// TIA Portal V19 export
ORGANIZATION_BLOCK "RESTART"   // OB100, STL, Startup
TITLE = Start-Up
{ S7_Optimized_Access := 'TRUE' }
VERSION : 0.0
// Comment
// stored: AutoNumber false
   VAR_INPUT
      LostRetentive : Bool;   // True if retentive data are lost
      LostRTC : Bool;   // True if date and time are lost
   END_VAR
BEGIN

NETWORK
TITLE = 
      L     0;
      T     "OP25 TANK".TaTimerStep;
      T     "OP25 TANK".TaTimerActual;
      T     "OP25 TANK".TaMainUpdating;
      T     "OP25 TANK".TaStepUpdating;

NETWORK
TITLE = 
      SET;
      R     "LEDAssignment".K1_FLASH;  //"FLASH_K1_SPARE"
      R     "LEDAssignment".K1_LIGHT;  //"LIGHT_K1_SPARE"
      R     "LEDAssignment".K2_FLASH;  //"FLASH_K2_SPARE"
      R     "LEDAssignment".K2_LIGHT;  //"LIGHT_K2_SPARE"
      R     "LEDAssignment".K3_FLASH;  //"FLASH_K3_PRESTE."
      R     "LEDAssignment".K3_LIGHT;  //"LIGHT_K3_PRESTE."
      R     "LEDAssignment".K4_FLASH;  //"FLASH_K4_CIP_LYE"
      R     "LEDAssignment".K4_LIGHT;  //"LIGHT_K4_CIP_LYE"
      R     "LEDAssignment".K5_FLASH;  //"FLASH_K5_CIP_LYE_ACID"
      R     "LEDAssignment".K5_LIGHT;  //"LIGHT_K5_CIP_LYE_ACID"
      R     "LEDAssignment".K6_FLASH;  //"FLASH_K6_DRAIN_TANK"
      R     "LEDAssignment".K6_LIGHT;  //"LIGHT_K6_DRAIN_TANK"
      R     "LEDAssignment".K7_FLASH;  //"FLASH_K7_STOP"
      R     "LEDAssignment".K7_LIGHT;  //"LIGHT_K7_STOP"




NETWORK
TITLE = initialise M0940 PID Loop setting for Pressure Control
      L     "M0940_PIDInterfaceDB".PC.P;
      T     "PIDHmiInterfaceDB".M0940.P;

      L     "M0940_PIDInterfaceDB".PC.I;
      T     "PIDHmiInterfaceDB".M0940.I;

      L     "M0940_PIDInterfaceDB".PC.D;
      T     "PIDHmiInterfaceDB".M0940.D;

      L     "M0940_PIDInterfaceDB".PC.SP;
      T     "PIDHmiInterfaceDB".M0940.SP;

      L     "M0940_PIDInterfaceDB".PC.EngUnitsMin;
      T     "PIDHmiInterfaceDB".M0940.EngUnitsMin;

      L     "M0940_PIDInterfaceDB".PC.EngUnitsMax;
      T     "PIDHmiInterfaceDB".M0940.EngUnitsMax;


END_ORGANIZATION_BLOCK
